FUNCTION_BLOCK AdsReadVariable
VAR_INPUT
	NetID: STRING := '';
	Name: STRING;
	EN: BOOL;
	Destination: PVOID;
END_VAR
VAR_OUTPUT
	ENO: BOOL;
END_VAR
VAR
	PLC_ReadSymInfoByName: PLC_ReadSymInfoByName;
	ADSREADEX: ADSREADEX;
	State : INT := 0;
END_VAR

CASE State OF
0:
	IF EN THEN
		State := 1;
	END_IF
1:	
	PLC_ReadSymInfoByName(
		NETID := NetID, 
		PORT := 851, 
		SYMNAME := Name,
		TMOUT := T#5S,
		START := TRUE
	);
	State := 2;
2:
	PLC_ReadSymInfoByName();
	IF NOT PLC_ReadSymInfoByName.BUSY THEN
		PLC_ReadSymInfoByName(START := FALSE);
		ADSREADEX(
			NETID:= '',
			PORT:= 851,
			IDXGRP:= PLC_ReadSymInfoByName.SYMINFO.idxGroup,
			IDXOFFS:= PLC_ReadSymInfoByName.SYMINFO.idxOffset,
			LEN:= SIZEOF(PLC_ReadSymInfoByName.SYMINFO.byteSize),
			DESTADDR:= Destination,
			READ:= TRUE,
			TMOUT:= T#5S,
		);
		State := 3;		
	END_IF
	IF NOT EN THEN
		ADSREADEX(READ := FALSE);
		ENO := FALSE;
		State := 0;
	END_IF
3:
	ADSREADEX();
	IF NOT ADSREADEX.BUSY THEN
		ENO := TRUE;
		ADSREADEX(READ := FALSE);
	END_IF
	IF NOT EN THEN
		ADSREADEX(READ := FALSE);
		ENO := FALSE;
		State := 0;
	END_IF
END_CASE

END_FUNCTION_BLOCK

(* stored: Version 1.1.0.1, ProductVersion 3.1.4024.6
   POU AdsReadVariable: Id {1b130b30-5abe-491f-8325-bcb8d0067140}, SpecialFunc None *)
